PROGRAM Axis03_Interlock
VAR
	Always_ON	:	BOOL	:=TRUE	;//상시 ON 
	Always_OFF	:	BOOL	:=FALSE	;//상시 OFF
END_VAR
VAR // added by the converter: edge detectors and wires of the graphical bodies
    _w1, _w2 : BOOL;
END_VAR

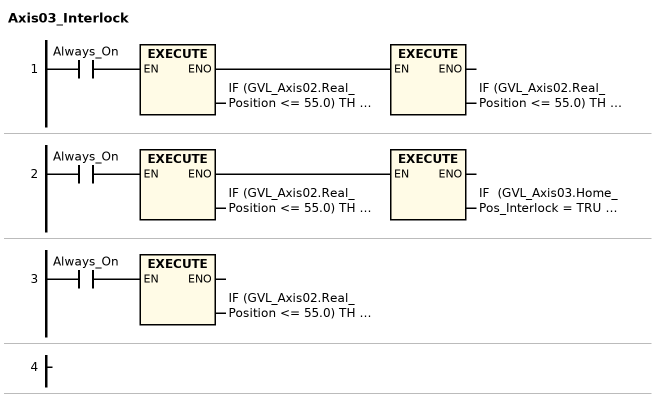
// NETWORK 1
_w1 := Always_On;
IF _w1 THEN
    IF (GVL_Axis02.Real_Position <= 55.0) THEN
        GVL_Axis03.Home_Pos_Interlock := TRUE;
    ELSE
        IF (GVL_Axis03.Home_Position_Data >= 3.4) AND 
           (GVL_Axis03.Home_Position_Data <= 48) THEN
            GVL_Axis03.Home_Pos_Interlock := TRUE;
        ELSE 
           GVL_Axis03.Home_Pos_Interlock := FALSE;
        END_IF;
    END_IF;
END_IF
IF _w1 THEN
    IF (GVL_Axis02.Real_Position <= 55.0) THEN
        GVL_Axis03.Wait_Pos_Interlock := TRUE;
    ELSE
        IF (GVL_Axis03.Wait_Position_Data >= 3.4) AND 
           (GVL_Axis03.Wait_Position_Data <= 48) THEN
           GVL_Axis03.Wait_Pos_Interlock := TRUE;
        ELSE 
           GVL_Axis03.Wait_Pos_Interlock := FALSE;
        END_IF;
    END_IF;
END_IF

// NETWORK 2
_w2 := Always_On;
IF _w2 THEN
    IF (GVL_Axis02.Real_Position <= 55.0) THEN
        GVL_Axis03.Work_End_Pos_Interlock := TRUE;
    ELSE
        IF (GVL_Axis03.Work_End_Position_Data >= 3.4) AND 
           (GVL_Axis03.Work_End_Position_Data <= 48) THEN
            GVL_Axis03.Work_End_Pos_Interlock := TRUE;
        ELSE 
           GVL_Axis03.Work_End_Pos_Interlock := FALSE;
        END_IF;
    END_IF;
END_IF
IF _w2 THEN
    IF  (GVL_Axis03.Home_Pos_Interlock = TRUE)
    AND (GVL_Axis03.Wait_Pos_Interlock = TRUE) AND (GVL_Axis03.Work_End_POs_Interlock = TRUE) THEN
    	GVL_Axis03.Interlock := TRUE;
    	ELSE
    	GVL_Axis03.Interlock := FALSE;	
    
    END_IF
END_IF

// NETWORK 3
IF Always_On THEN
    IF (GVL_Axis02.Real_Position <= 55.0) THEN
        GVL_Axis03.Home_ORG_Interlock := TRUE;
    ELSE
        GVL_Axis03.Home_ORG_Interlock := FALSE;
    
    END_IF;
END_IF

// NETWORK 4

END_PROGRAM

(* stored: Version 1.1.0.1, ProductVersion 3.1.4024.15
   POU Axis03_Interlock: Id {55902515-fa66-4c8c-b0c4-11bac34c4f15}, SpecialFunc None *)
